FUNCTION_BLOCK FB_PcSafeOff
VAR
	fbWritePersistentData		:FB_WritePersistentData;
	fbPlcStop					:PLC_Stop;
	fbNtShutdown				:NT_Shutdown;
	fbNtReboot					:NT_Reboot;
	
	PcAmsNetId					:AMSNETID;					//PC AMS Net ID
	
	fbRebootTon					:TON;
	fbShutdownTon				:TON;
	
	iRebootStep					:INT;
	iShutdownStep				:INT;
END_VAR

//FB_Init は常に暗黙的に使用可能で、主に初期化に使用されます。
//戻り値は評価されません。特定の結果を得るために、メソッドを明示的に宣言し、
//そのメソッドに標準の初期化コードをもったコードを追加することができます。戻り値を評価できます。
METHOD FB_Init: BOOL
VAR_INPUT
    bInitRetains: BOOL; // TRUE: 保持変数は初期化されます (ウォーム リセット、あるいはコールド リセット)
    bInCopyCode: BOOL;  // TRUE: 後でコードをコピーする (オンライン変更) ために、インスタンスをコピーします。

	PcAmsNetId			:AMSNETID;		//PC AMS Net ID
END_VAR
THIS^.PcAmsNetId		:=PcAmsNetId;
END_METHOD

METHOD Reboot
VAR_INPUT
	bReboot	:bool;
END_VAR
CASE iRebootStep OF
	0:
		fbRebootTon(IN:=bReboot,PT:=T#2S,Q=>,ET=>);
			
		IF fbRebootTon.Q=TRUE THEN
			fbWritePersistentData.START:=TRUE;
			iRebootStep:=1;			
		END_IF

	1:
		fbWritePersistentData(	NETID	:=F_CreateAmsNetId(PcAmsNetId),
								PORT	:=_AppInfo.AdsPort,
								START	:=,
								TMOUT	:=DEFAULT_ADS_TIMEOUT,
								MODE	:=E_PersistentMode.SPDM_2PASS,
								BUSY	=>,
								ERR		=>,
								ERRID	=>
								);
	
		IF fbWritePersistentData.BUSY=FALSE THEN
			fbWritePersistentData.START:=FALSE;
			iRebootStep:=2;
		END_IF
	
	2:
		fbPlcStop.STOP:=TRUE;
		fbNtReboot.START:=TRUE;
		iRebootStep:=3;
	
	3:
		fbPlcStop(	NETID	:=F_CreateAmsNetId(PcAmsNetId),
					PORT	:=_AppInfo.AdsPort,
					Stop	:=,
					TMOUT	:=DEFAULT_ADS_TIMEOUT,
					BUSY	=>,
					ERR		=>,
					ERRID	=>
					);

		fbNtReboot(	NETID	:=F_CreateAmsNetId(PcAmsNetId),
					DELAY	:=1,
					START	:=,
					TMOUT	:=DEFAULT_ADS_TIMEOUT,
					BUSY	=>,
					ERR		=>,
					ERRID	=>
					);

END_CASE
END_METHOD

METHOD Shutdown
VAR_INPUT
	bShutdown	:BOOL;
END_VAR
CASE iShutdownStep OF
	0:
		fbShutdownTon(IN:=bShutdown,PT:=T#2S,Q=>,ET=>);
	
		IF fbShutdownTon.Q=TRUE THEN
			fbWritePersistentData.START:=TRUE;
			iShutdownStep:=1;			
		END_IF

	1:
		fbWritePersistentData(	NETID	:=F_CreateAmsNetId(PcAmsNetId),
								PORT	:=_AppInfo.AdsPort,
								START	:=,
								TMOUT	:=DEFAULT_ADS_TIMEOUT,
								MODE	:=E_PersistentMode.SPDM_2PASS,
								BUSY	=>,
								ERR		=>,
								ERRID	=>
								);
	
		IF fbWritePersistentData.BUSY=FALSE THEN
			fbWritePersistentData.START:=FALSE;
			iShutdownStep:=2;
		END_IF
	
	2:
		fbPlcStop.STOP:=TRUE;
		fbNtShutdown.START:=TRUE;
		iShutdownStep:=3;
	
	3:
		fbPlcStop(	NETID	:=F_CreateAmsNetId(PcAmsNetId),
					PORT	:=_AppInfo.AdsPort,
					Stop	:=,
					TMOUT	:=DEFAULT_ADS_TIMEOUT,
					BUSY	=>,
					ERR		=>,
					ERRID	=>
					);

		fbNtShutdown(	NETID	:=F_CreateAmsNetId(PcAmsNetId),
						DELAY	:=1,
						START	:=,
						TMOUT	:=DEFAULT_ADS_TIMEOUT,
						BUSY	=>,
						ERR		=>,
						ERRID	=>
						);
	
END_CASE
END_METHOD

END_FUNCTION_BLOCK

(* stored: Version 1.1.0.1, ProductVersion 3.1.4026.11
   POU FB_PcSafeOff: Id {a838037a-1898-4803-a40b-4cae93a39ef4}, SpecialFunc None
   Method FB_Init: Id {9ffa7f8d-2ee0-4b92-b303-254ac03ae195}
   Method Reboot: Id {d1d1267f-1e25-4cdd-ab44-1fe5180ef081}
   Method Shutdown: Id {b0d0c740-c26b-4bb4-9fc2-86d7cf6edd45} *)
